(* LS Electric XG5000 project: Study2_Functions *)
(* PLC LSPLC *)
(* module base 0 slot 0: 입력 모듈:XGI-D21A (DC 24V 입력, 8점 (전류소스/싱크입력)) *)
(* module base 0 slot 1: 출력 모듈:XGQ-RY1A (릴레이 출력, 8점 (2A용, 단독 COM.)) *)

PROGRAM NewProgram (* task: 스캔 프로그램 *)
VAR
    data1 : INT;
    data2 : INT;
    data3 : INT;
    data4 : INT;
    data5 : INT;
    data6 : INT;
    data7 : INT;
    data8 : INT;
    output1 : INT;
    output2 : INT;
    output3 : INT;
    output4 : INT;
    outputout : INT;
    램프1 AT %QX0.1.2 : BOOL;
    램프2 AT %QX0.1.1 : BOOL;
    타이머1 : TON;
    타이머2 : TON;
END_VAR

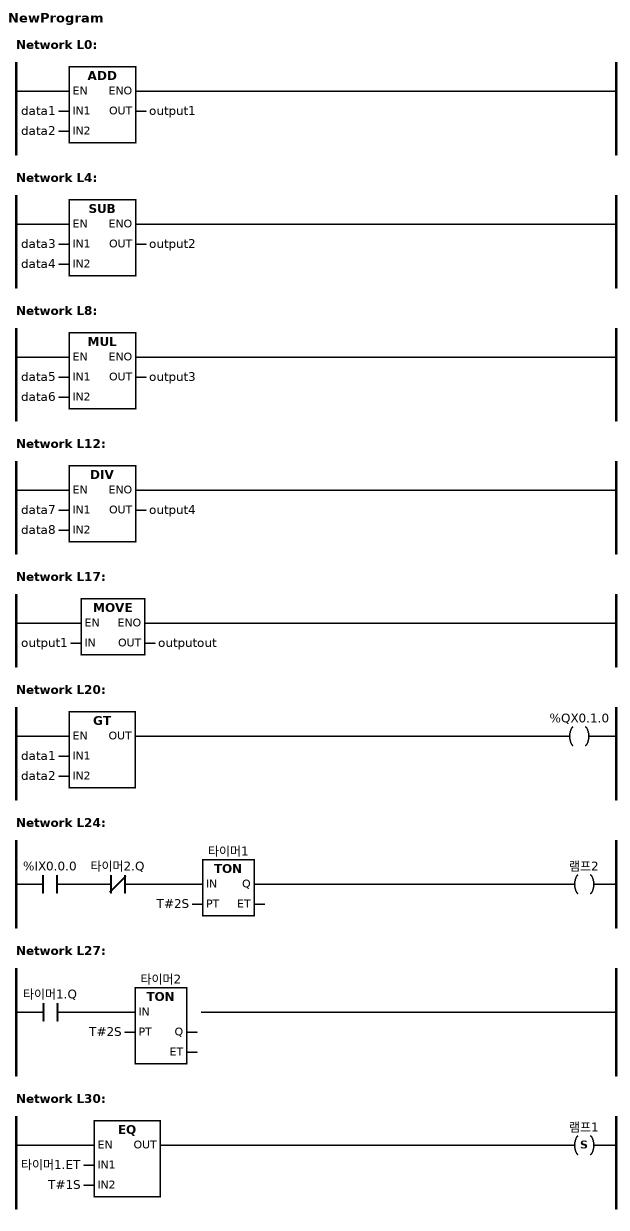
(* Rung L0 *)
output1 := data1 + data2;
(* Rung L4 *)
output2 := data3 - data4;
(* Rung L8 *)
output3 := data5 * data6;
(* Rung L12 *)
output4 := data7 / data8;
(* Rung L17 *)
outputout := output1;
(* Rung L20 *)
%QX0.1.0 := data1 > data2;
(* Rung L24 *)
타이머1(IN := %IX0.0.0 AND NOT 타이머2.Q, PT := T#2S);
램프2 := 타이머1.Q;
(* Rung L27 *)
타이머2(IN := 타이머1.Q, PT := T#2S);
(* Rung L30 *)
IF 타이머1.ET = T#1S THEN 램프1 := TRUE; END_IF;
END_PROGRAM